FUNCTION_BLOCK INTERNAL FB_WaitingState IMPLEMENTS I_State
VAR_INPUT
END_VAR
VAR_OUTPUT
END_VAR
VAR
	pMachine : I_StateMachine;
	coinInsertedNext : I_State;
END_VAR

METHOD CustomerTakesCoin : BOOL
END_METHOD

METHOD CustomerTakesProduct : BOOL
END_METHOD

PROPERTY Description : STRING
GET
Description := 'Waiting';
END_GET
END_PROPERTY

METHOD InsertCoin : BOOL
ADSLOGSTR(ADSLOG_MSGTYPE_HINT, 'Customer has insert a coin.', '');
pMachine.SetState(coinInsertedNext);
END_METHOD

METHOD PressButton : BOOL
END_METHOD

METHOD SetTransitionStates
VAR_INPUT
	Machine : I_StateMachine;
	CoinInsertedNext : I_State;
END_VAR
THIS^.coinInsertedNext := CoinInsertedNext;
THIS^.pMachine := Machine;
END_METHOD

END_FUNCTION_BLOCK

(* stored: Version 1.1.0.1, ProductVersion 3.1.4022.17
   POU FB_WaitingState: Id {bcf41680-3dab-4cd9-bc56-3d8d89453988}, SpecialFunc None
   Method CustomerTakesCoin: Id {76b1ff06-f114-4365-8fa1-73ab525d2621}
   Method CustomerTakesProduct: Id {9a03121f-9796-4862-9404-a52a1e9ee2e9}
   Property Description: Id {b13bfef9-dadc-4c1e-bb5d-4339f02951be}
   Get Get: Id {517ae1c8-c5a2-4678-b562-7b6f58d256eb}
   Method InsertCoin: Id {f8f4dc73-5d56-4b22-a640-25d47afc33d7}
   Method PressButton: Id {291ec246-7036-4eab-8c64-3c8ae17a9320}
   Method SetTransitionStates: Id {44d6c76c-96c0-49c2-a953-8ae130620548} *)
